// TIA Portal V20 export
TYPE "s_zc_NormalInterlocks"
// stored: Access Published, IsFailsafeCompliant true, Namespace Safety
   STRUCT
      AutorunMode { ExternalWritable := 'False'} : Bool := FALSE;   // Auto mode is selected on select button and OMAC is on production mode.
      ManualMode { ExternalWritable := 'False'} : Bool := FALSE;   // Auto mode is selected on select button and OMAC is on manual mode.
      SCS_AutoMode : Bool;
      SCS_SetupMode { ExternalWritable := 'False'} : Bool := FALSE;   // Setup mode is selected on select button and OMAC is on maintenance mode.
      SCS_DisableMode { ExternalWritable := 'False'} : Bool := FALSE;   // Disable mode is selected.
      TestStopComplete { ExternalWritable := 'False'} : Bool := FALSE;   // All safety test are completed on vertical axes.
      TestStopActivated { ExternalWritable := 'False'} : Bool := FALSE;   // Any safety test is activated on vertical axis.
      NoInterference { ExternalWritable := 'False'} : Bool := FALSE;   // No interference in loading/unloading area.
      NotCollisionArea { ExternalWritable := 'False'} : Bool := FALSE;   // Ack. interference area since finish the loading/unloading.
      reserved00 { ExternalWritable := 'False'} : Bool := FALSE;   // Ack. interference area since finish the loading/unloading.
      reserved01 { ExternalWritable := 'False'} : Bool := FALSE;   // reserved
      reserved02 { ExternalWritable := 'False'} : Bool := FALSE;   // reserved
      reserved03 { ExternalWritable := 'False'} : Bool := FALSE;   // reserved
      reserved04 { ExternalWritable := 'False'} : Bool := FALSE;   // reserved
      reserved05 { ExternalWritable := 'False'} : Bool := FALSE;   // reserved
      reserved06 { ExternalWritable := 'False'} : Bool := FALSE;   // reserved
      reserved07 { ExternalWritable := 'False'} : Bool := FALSE;   // reserved
      reserved08 { ExternalWritable := 'False'} : Bool := FALSE;   // reserved
      reserved09 { ExternalWritable := 'False'} : Bool := FALSE;   // reserved
      reserved10 { ExternalWritable := 'False'} : Bool;
      reserved11 { ExternalWritable := 'False'} : Bool;
      reserved12 { ExternalWritable := 'False'} : Bool;
      reserved13 { ExternalWritable := 'False'} : Bool;
      reserved14 { ExternalWritable := 'False'} : Bool;
      reserved15 { ExternalWritable := 'False'} : Bool;
      reserved16 { ExternalWritable := 'False'} : Bool;
      reserved17 { ExternalWritable := 'False'} : Bool;
      reserved18 { ExternalWritable := 'False'} : Bool;
      reserved19 { ExternalWritable := 'False'} : Bool;
      reserved20 { ExternalWritable := 'False'} : Bool;
      reserved21 { ExternalWritable := 'False'} : Bool;
      reserved22 { ExternalWritable := 'False'} : Bool;
   END_STRUCT;
END_TYPE
